FUNCTION_BLOCK EM_AirTreatment EXTENDS EM_Base IMPLEMENTS I_EM_AirTreatment
VAR_INPUT
END_VAR
VAR_OUTPUT
END_VAR
VAR
END_VAR

METHOD PUBLIC m_Equalize : BOOL
END_METHOD

METHOD PUBLIC m_Flush : BOOL
END_METHOD

METHOD PUBLIC m_Pressurize : BOOL
END_METHOD

PROPERTY PUBLIC p_bStaEqualizingDone : BOOL
GET
END_GET
END_PROPERTY

PROPERTY PUBLIC p_bStaFlushingDone : BOOL
GET
END_GET
END_PROPERTY

PROPERTY PUBLIC p_bStaPressurizingOK : BOOL
GET
END_GET
END_PROPERTY

END_FUNCTION_BLOCK

(* stored: Version 1.1.0.1, ProductVersion 3.1.4024.12
   POU EM_AirTreatment: Id {81e48a97-313d-405f-b257-49532a716bbe}, SpecialFunc None
   Method m_Equalize: Id {3dbf5f0e-de32-4d1f-a1ee-f80454ebc838}
   Method m_Flush: Id {91abc485-ede4-4dc8-9260-f53c4f914a84}
   Method m_Pressurize: Id {7248c420-f75f-49e3-bdd0-b32fa28f9dd2}
   Property p_bStaEqualizingDone: Id {70485294-9ae5-46f7-b455-a30567b2984d}
   Get Get: Id {512491e2-2c43-4c65-af17-560f948bfa0e}
   Property p_bStaFlushingDone: Id {e8505bce-20c5-4e11-a93c-d9c8bb05b3bb}
   Get Get: Id {56be4fba-47da-4dfb-819b-1e2798cd877e}
   Property p_bStaPressurizingOK: Id {7ff7c161-f01c-480d-8d30-a3ec8426337a}
   Get Get: Id {a6f3a68e-e97d-4c33-8765-cf3f9408337e} *)
